// TIA Portal V18 export
// export: Created 2026-01-09T11:32:10.0107368Z, ExportSetting WithDefaults, DisplayName Totally Integrated Automation Portal, DisplayVersion V18 Update 5, DisplayName TIA Portal Openness, DisplayVersion V18 Update 5, DisplayName TIA Portal Teamcenter Gateway, DisplayVersion V18, DisplayName TIA Portal Version Control Interface, DisplayVersion V18, DisplayName SINAMICS Startdrive Advanced, DisplayVersion V18 SP2 Update 1, DisplayName SINAMICS Startdrive G110M, G120, G120C, G120D, G120P, G115D, DisplayVersion V18 SP2 Update 1, DisplayName SINAMICS Startdrive G130, G150, S120, S150, SINAMICS MV, S210, G220, S200, DisplayVersion V18 SP2 Update 1, DisplayName STEP 7 Professional, DisplayVersion V18 Update 5, DisplayName STEP 7 Safety, DisplayVersion V18, DisplayName WinCC Professional, DisplayVersion V18 Update 5
TagTable "IAI"
  HMISystemDB_HMI_Axis : HMI_Axis  (PLC tag HMISystemDB.HMI_Axis, CPU S71500-2PN_TP700, 1 s)
    TagStructureMember "INPUT"
      TagStructureMember "Axis_ID"
      TagStructureMember "Speed"
      TagStructureMember "SimplyTrigger"
      TagStructureMember "ListTrigger"
      TagStructureMember "ListPosID"
      TagStructureMember "SimplyPos"
      TagStructureMember "Enable"
      TagStructureMember "Jog+"
      TagStructureMember "Jog-"
      TagStructureMember "Homing"
      TagStructureMember "Stop"
    TagStructureMember "OUTPUT"
      TagStructureMember "Ready"
      TagStructureMember "Alarm"
      TagStructureMember "Warming"
      TagStructureMember "RunEnd"
      TagStructureMember "Interference"
      TagStructureMember "Reference Point"
      TagStructureMember "CurrentPosition"
      TagStructureMember "CurrentSpeed"
      TagStructureMember "TargetPosition"
      TagStructureMember "Enable"
      TagStructureMember "MAX_Axis"
